// TIA Portal V20 export
TYPE "typeFDoorSignal"
// Safety status of door
// stored: Access Published, IsFailsafeCompliant true, Namespace Safety
   STRUCT
      reqDoorUnlock1 : Bool;   // Cmd Maint Door1 Open Request
      reqDoorUnlock2 : Bool;   // Cmd Maint Door2 Open Request
      reqDoorUnlock6 : Bool;   // Cmd Maint Door6 Open Request
      reqDoorUnlock7 : Bool;   // Cmd Maint Door7 Open Request
   END_STRUCT;
END_TYPE
